Universal Robots PolyScope program: 22-thread.urp

ProgramRoot directory=/home/ur/ursim-3.1/programs/basic training/22-thread; kinematics=(a=[0, -0.425, -0.39225, 0, 0, 0], d=[0.08916, 0, 0, 0.10915, 0.09465, 0.0823], alpha=[1.5708, 0, 0, 1.5708, -1.5708, 0], deltaTheta=[0, 0, 0, 0, 0, 0], status=notInitialized); lastSavedInVersion=(project__name=Polyscope, major__version=3, minor__version=1, svn__revision=17195, build__date=Mar 11 2015, 13:02:28); name=22-thread; programVersion=(project__name=Polyscope, major__version=3, minor__version=1, svn__revision=17195, build__date=Mar 11 2015, 13:02:28); robotEnvironmentFileName=default; serialNumberRobot=2014350001
  MainProgram cartesianAcceleration=1.2; cartesianSpeed=0.25; jointAcceleration=1.3962634015954636; jointSpeed=1.0471975511965976; sharedProcessMoveBlendRadius=0.025; motionType=JOINT_SPACE
    Move cartesianAcceleration=1.2; cartesianSpeed=0.25; jointAcceleration=1.3962634015954636; jointSpeed=1.0471975511965976; sharedProcessMoveBlendRadius=0.025; motionType=JOINT_SPACE
      Waypoint blendRadius=0.05; cartesianAcceleration=1.2; cartesianSpeed=0.25; jointAcceleration=1.3962634015954636; jointSpeed=1.0471975511965976; nextMotionTime=2.0; stoppoint=true; useSharedBlendParameter=true; useSharedParameters=true; position=TCP in base x=313.816 y=-411.952 z=426.714 mm, rx=-0.0012 ry=3.1163 rz=0.0389 rad; joints [-40.862, -92.666, -88.063, -89.122, 92.021, 49.096] deg; positionType=FIXED_POSITION; waypointPoseInFeatureCoordinates=(pos=(x=0.31381590983180896, y=-0.4119516485752222, z=0.42671398574289104), rot=(x=-0.0012210227574820896, y=3.1162763421843955, z=0.03889217574521001)); name=路点_2
      Waypoint blendRadius=0.05; cartesianAcceleration=1.2; cartesianSpeed=0.25; jointAcceleration=1.3962634015954636; jointSpeed=1.0471975511965976; nextMotionTime=2.0; stoppoint=true; useSharedBlendParameter=true; useSharedParameters=true; position=TCP in base x=313.816 y=-411.952 z=179.895 mm, rx=-0.0012 ry=3.1163 rz=0.0389 rad; joints [-40.862, -103.84, -113.869, -52.14, 92.021, 49.096] deg; positionType=FIXED_POSITION; waypointPoseInFeatureCoordinates=(pos=(x=0.3138159317220093, y=-0.4119516674444875, z=0.17989535093785725), rot=(x=-0.0012210227574801476, y=3.1162763421843898, z=0.03889217574521966)); name=路点_1
  Thread name=线程_1
    If expr=ExpressionIONode; type=IF_NODE
      Halt 
    Script type=0; expressionBranchNode=sync()
